(* PLC project light, Dassault Systèmes ControlBuild 2024x *)
(* stored: creationDateTime 2023-10-03T11:13:24-01:00 *)

(* This module simulates a light. *)
FUNCTION_BLOCK equipment_library.light
  VAR_INPUT
    luminous : BOOL := false;
  END_VAR

(* -----------------------------------------------------------------	*)
(* Type : Model of Operative Behaviour					*)
(* Category :  Power								*)
(* Author : Dassault Systemes						*)
(* Update date : June 2010							*)
(* -----------------------------------------------------------------	*)
(* This module simulates a light.				 		*)
(* -----------------------------------------------------------------	*)
END_FUNCTION_BLOCK
